// TwinCAT 3 PLC project PLC_Project
// ProgramVersion: 3.1.4023.0
// libraries:
//   Tc2_Standard, * (Beckhoff Automation GmbH)
//   Tc2_System, * (Beckhoff Automation GmbH)
//   Tc3_Module, * (Beckhoff Automation GmbH)
// project tree:
//   / PlcTask.TcTTO
//   POUs/ FB_PULSO.TcPOU, MAIN.TcPOU, Main_PULSO.TcPOU, POU.TcPOU, References.TcPOU
// real-time tasks:
//   TASK PlcTask: cycle T#10ms, priority 20, ADS port 350
//   TASK PlcTask1: cycle T#10ms, priority 21, ADS port 351
// motion (NC):
//   TASK NC-Task 1 SAF: cycle T#2ms, priority 4, ADS port 501
//   TASK NC-Task 1 SVB: cycle T#10ms, priority 8, ADS port 511
//   AXIS Axis 1 (id 1)
//     OtherSettings: AllowMotionCmdToSlave=true
//     encoder EncType=1
//     drive DrvType=5
//       Analog: VeloReferenz=4400, TorqueSetpointScale=10, ScaleFactorActTorque=0.1
//       TimeComp: TaskDelayCycles=1
//     controller CtrType=1
//       CtrPara: PriorControlFactor=1
//         Observer: BandWidth=20
//   AXIS Axis 2 (id 2)
//     OtherSettings: AllowMotionCmdToSlave=true
//     encoder EncType=1
//     drive DrvType=5
//       Analog: VeloReferenz=3000, TorqueSetpointScale=10, ScaleFactorActTorque=0.1
//       TimeComp: TaskDelayCycles=1
//     controller CtrType=1
//       CtrPara: PriorControlFactor=1
//         Observer: BandWidth=20
// I/O:
//   DEVICE Device 1 (EtherCAT), AmsNetId 192.168.1.37.2.1
//     Term 1 (EK1100) [EK1100 EtherCAT Coupler (2A E-Bus)]
//       Term 3 (EL1004) [EL1004 4Ch. Dig. Input 24V, 3ms]
//     Box 2 (EP2318-0001) [EP2318-0001 4 Ch. Dig. In, 10µs, 4 Ch. Dig. Out 24V, 0,5A, M8]
// variable links:
//   PLC_Project Instance <-> Device 1 (EtherCAT)/Box 2 (EP2318-0001)
//     PlcTask Inputs/MAIN.VarIn <-> Channel 1/Input
//     PlcTask Outputs/MAIN.VarOut <-> Channel 5/Output
//     PlcTask Outputs/MAIN.VarOut2 <-> Channel 6/Output
//   PLC_Project Instance <-> Device 1 (EtherCAT)/Term 1 (EK1100)/Term 3 (EL1004)
//     PlcTask Inputs/MAIN.VarIn2 <-> Channel 2/Input

CONFIGURATION PLC_Project
    RESOURCE PLC ON TwinCAT3
        TASK PlcTask(INTERVAL := T#10ms, PRIORITY := 21);
        PROGRAM MAIN WITH PlcTask : MAIN;
    END_RESOURCE
END_CONFIGURATION

// ---- POUs/MAIN.TcPOU
PROGRAM MAIN
VAR
	VarOut AT %Q*: BOOL;
	VarIn AT %I*: BOOL;
	VarOut2 AT %Q*: BOOL;
	VarIn2 AT %I*: BOOL;
	Paso: INT;
	SALTO_A_30: BOOL;

	SALTO_A_10: BOOL;
END_VAR

// Comentario
Cambios a las 0:11
     //ADSLOGDINT(msgCtrlMask:= ADSLOG_MSGTYPE_LOG, msgFmtStr := 'PLC Msg: Feed too high! Current feed: %d', dintArg := Paso);
 ADSLOGDINT(msgCtrlMask:= ADSLOG_MSGTYPE_LOG, msgFmtStr := 'Paso Actual: %d', dintArg := Paso);
CASE Paso OF
	10:
     ADSLOGSTR(msgCtrlMask:= ADSLOG_MSGTYPE_LOG, msgFmtStr := 'EN PASO 10' , strArg := ' '); 
     Paso := 20;
	
	20:
	
	 IF SALTO_A_30 THEN
		 ADSLOGSTR(msgCtrlMask:= ADSLOG_MSGTYPE_LOG, msgFmtStr := 'SALTO A 30' , strArg := ' ');
		 Paso := 30;
	 END_IF
	  IF SALTO_A_10 THEN
		 ADSLOGSTR(msgCtrlMask:= ADSLOG_MSGTYPE_LOG, msgFmtStr := 'SALTO A 10' , strArg := ' ');
		 Paso := 10;
	  ELSE
	      ADSLOGSTR(msgCtrlMask:= ADSLOG_MSGTYPE_LOG, msgFmtStr := 'ELSE PASO 20' , strArg := ' ');
		  END_IF
		   
	30:
	     ADSLOGSTR(msgCtrlMask:= ADSLOG_MSGTYPE_LOG, msgFmtStr := 'EN PASO 30' , strArg := ' ');
END_CASE

END_PROGRAM

// ---- POUs/FB_PULSO.TcPOU
FUNCTION_BLOCK FB_PULSO
VAR_INPUT
	Referencia_a_variable_a_Pulsar: REFERENCE TO BOOL;
	Temps_pols : TIME;	
END_VAR
VAR_OUTPUT

END_VAR
VAR
	TP1: TP;
	Activar_TP1 : BOOL;
	Temps : TIME;
	Temps_actual_pols : TIME;
	Variable_pulsdada : BOOL;
END_VAR

   



     TP1(IN:= Referencia_a_variable_a_Pulsar , PT:=  Temps_pols, Q=> Variable_pulsdada   , ET=> Temps_actual_pols  );
	IF TP1.ET = TP1.PT THEN Referencia_a_variable_a_Pulsar := FALSE ;
		// <
	END_IF

END_FUNCTION_BLOCK

// ---- POUs/Main_PULSO.TcPOU
PROGRAM Main_PULSO
// HAY QUE HACER UN OBJETO DE CADA FUNCTION BLOCK PARA CADA VARIABLE
VAR
	Variable_a_pulsar: BOOL;
	Variable_a_pulsar_1: BOOL;
	FB_PULSO_1: FB_PULSO;
	paso: INT;
	FB_PULSO_2: FB_PULSO;
END_VAR

//ADSLOGDINT(msgCtrlMask:= ADSLOG_MSGTYPE_LOG, msgFmtStr := 'Paso Actual Inicio: %d', dintArg := Paso);

CASE paso  OF


10:
//IF Variable_a_pulsar = TRUE THEN  
	FB_PULSO_1(Referencia_a_variable_a_Pulsar := Variable_a_pulsar , Temps_pols := T#4S );
	ADSLOGDINT(msgCtrlMask:= ADSLOG_MSGTYPE_LOG, msgFmtStr := 'Paso Actual 10: %d', dintArg := Paso);
	FB_PULSO_2(Referencia_a_variable_a_Pulsar := Variable_a_pulsar_1, Temps_pols := T#10S );
//END_IF

//paso := 20;

20:
FB_PULSO_1(Referencia_a_variable_a_Pulsar := Variable_a_pulsar , Temps_pols := T#4S );    	
// FB_PULSO_1(Referencia_a_variable_a_Pulsar := Variable_a_pulsar_1 , Temps_pols := T#4S );
//ADSLOGDINT(msgCtrlMask:= ADSLOG_MSGTYPE_LOG, msgFmtStr := 'Paso Actual 20: %d', dintArg := Paso);

END_CASE

END_PROGRAM

// ---- POUs/POU.TcPOU
PROGRAM POU
VAR
	Paso: INT;
	SALTO_A_30: BOOL;
	SALTO_A_10: BOOL;	
	SALTO_A_20: BOOL;	

	Trans0: BOOL;
	VarOut AT %Q*: BOOL;
	VarIn AT %I*: BOOL;
	VarOut2 AT %Q*: BOOL;
	VarIn2 AT %I*: BOOL;
END_VAR

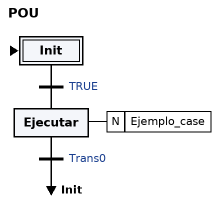
INITIAL_STEP Init:
END_STEP
TRANSITION FROM Init TO Ejecutar
    := TRUE;
END_TRANSITION
STEP Ejecutar:
    Ejemplo_case(N);
END_STEP
TRANSITION FROM Ejecutar TO Init
    := Trans0;
END_TRANSITION

ACTION Ejemplo_case:
     ADSLOGDINT(msgCtrlMask:= ADSLOG_MSGTYPE_LOG, msgFmtStr := 'Paso Actual: %d', dintArg := Paso);

CASE Paso OF
	10:
     ADSLOGSTR(msgCtrlMask:= ADSLOG_MSGTYPE_LOG, msgFmtStr := 'EN PASO 10' , strArg := ' '); 
     Paso := 20;
	
	20:
	
	 IF SALTO_A_30 THEN
		 ADSLOGSTR(msgCtrlMask:= ADSLOG_MSGTYPE_LOG, msgFmtStr := 'SALTO A 30' , strArg := ' ');
		 Paso := 30;
	 END_IF
	  IF SALTO_A_10 THEN
		 ADSLOGSTR(msgCtrlMask:= ADSLOG_MSGTYPE_LOG, msgFmtStr := 'SALTO A 10' , strArg := ' ');
		 Paso := 10;
	  ELSE
	      ADSLOGSTR(msgCtrlMask:= ADSLOG_MSGTYPE_LOG, msgFmtStr := 'ELSE PASO 20' , strArg := ' ');
		  END_IF
		   
	30:
	     ADSLOGSTR(msgCtrlMask:= ADSLOG_MSGTYPE_LOG, msgFmtStr := 'EN PASO 30' , strArg := ' ');
          IF SALTO_A_20 THEN
		 ADSLOGSTR(msgCtrlMask:= ADSLOG_MSGTYPE_LOG, msgFmtStr := 'SALTO A 30' , strArg := ' ');
		 Paso := 20;
		 END_IF

END_CASE
END_ACTION

END_PROGRAM

// ---- POUs/References.TcPOU
PROGRAM References
VAR
	nVar      : INT;
    refInt1   : REFERENCE TO INT;
    refInt2   : REFERENCE TO INT;
    bTestRef1 : BOOL := FALSE;
    bTestRef2 : BOOL := FALSE;
END_VAR

//nVar       := nVar + 1;
refInt1  REF= nVar;
refInt2  REF= 0;
//bTestRef1  := __ISVALIDREF(refInt1); (* becomes TRUE, because refInt1 points to nVar, which is non-zero *)
//bTestRef2  := __ISVALIDREF(refInt2); (* becomes FALSE, because refInt2 is set to 0 *)

END_PROGRAM
